// TIA Portal V20 export
VAR_GLOBAL   // PLC tag table "IMC88"
   IMC88Sensor_1 AT %I727.0 : Bool;   // High = Sensor active (input type and polarity can be configured)
   IMC88Sensor_2 AT %I727.1 : Bool;   // High = Sensor active (input type and polarity can be configured)
   IMC88Sensor_3 AT %I727.2 : Bool;   // High = Sensor active (input type and polarity can be configured)
   IMC88Sensor_4 AT %I727.3 : Bool;   // High = Sensor active (input type and polarity can be configured)
   IMC88Sensor_5 AT %I727.4 : Bool;
   IMC88Sensor_6 AT %I727.5 : Bool;
   IMC88Sensor_7 AT %I727.6 : Bool;
   IMC88Sensor_8 AT %I727.7 : Bool;
   IMC88IO1 AT %I728.0 : Bool;   // Digital I/O PLC Input PLC Output
   IMC88IO2 AT %I728.1 : Bool;   // Digital I/O PLC Input PLC Output
   IMC88IO3 AT %I728.2 : Bool;   // Digital I/O PLC Input PLC Output
   IMC88IO4 AT %I728.3 : Bool;   // Digital I/O PLC Input PLC Output
   IMC88IO5 AT %I728.4 : Bool;
   IMC88IO6 AT %I728.5 : Bool;
   IMC88IO7 AT %I728.6 : Bool;
   IMC88IO8 AT %I728.7 : Bool;
   "IMC88MotorStateErrorRD -G1.7.4" AT %I729.0 : Bool;   // High = Motor Error; Low = Motor OK
   "IMC88MotorStateErrorRD -G1.7.3" AT %I729.1 : Bool;   // High = Motor Error; Low = Motor OK
   "IMC88MotorStateErrorRD -G1.7.2" AT %I729.2 : Bool;   // High = Motor Error; Low = Motor OK
   "IMC88MotorStateErrorRD -4" AT %I729.3 : Bool;   // High = Motor Error; Low = Motor OK
   "IMC88MotorStateSpeedRD -G1.7.4" AT %IB730 : SInt;   // Speed 0–100 ( 0 = Stop, 100 = max speed), negative sign reverses the turning direction
   "IMC88MotorStateSpeedRD -G1.7.3" AT %IB731 : SInt;   // Speed 0–100 ( 0 = Stop, 100 = max speed), negative sign reverses the turning direction
   "IMC88MotorStateSpeedRD -G1.7.2" AT %IB732 : SInt;   // Speed 0–100 ( 0 = Stop, 100 = max speed), negative sign reverses the turning direction
   "IMC88MotorStateSpeedRD -4" AT %IB733 : SInt;   // Speed 0–100 ( 0 = Stop, 100 = max speed), negative sign reverses the turning direction
   "IMC88MotorCurrentRD -G1.7.4" AT %IW735 : Int;   // Average current in mA
   "IMC88MotorCurrentRD -G1.7.3" AT %IW737 : Int;   // Average current in mA
   "IMC88MotorCurrentRD -G1.7.2" AT %IW739 : Int;   // Average current in mA
   "IMC88MotorCurrentRD -4" AT %IW741 : Int;   // Average current in mA
   "IMC88Voltage(MotorPower)" AT %IW743 : Int;   // Voltage „Motor Power“ in mV
   "IMC88Voltage(Sensors)" AT %IW745 : Int;   // Voltage „Power Logic + Sensors“ in mV
   IMC88Temperature AT %IW747 : Int;   // Temperature in 0,1 C
   IMC88SystemUpTime AT %ID749 : DInt;   // Operating time in seconds since the last start/restart
   "IMC88DigitalOutputRD -G1.7.4" AT %Q535.0 : Bool;
   "IMC88DigitalOutputRD -G1.7.3" AT %Q535.1 : Bool;
   "IMC88DigitalOutputRD -G1.7.2" AT %Q535.2 : Bool;
   "IMC88DigitalOutputRD -4" AT %Q535.3 : Bool;
   "IMC88MotorTargetSpeedRD -G1.7.4" AT %QB536 : SInt;   // Speed 0–100 ( 0 = Stop, 100 = max speed), negative sign reverses the turning direction
   "IMC88MotorTargetSpeedRD -G1.7.3" AT %QB537 : SInt;   // Speed 0–100 ( 0 = Stop, 100 = max speed), negative sign reverses the turning direction
   "IMC88MotorTargetSpeedRD -G1.7.2" AT %QB538 : SInt;   // Speed 0–100 ( 0 = Stop, 100 = max speed), negative sign reverses the turning direction
   "IMC88MotorTargetSpeedRD -4" AT %QB539 : SInt;   // Speed 0–100 ( 0 = Stop, 100 = max speed), negative sign reverses the turning direction
END_VAR
